(* IEC 61131-3 sources: st2cpp/tests/st_samples, 5 files *)

(* ---- test_array.st ---- *)
// ============================================================================
// ENUM Definitions
// ============================================================================

TYPE Color :
    (
    Red,
    Green := 5,
    Blue,
    Yellow := 10
    );
END_TYPE

TYPE Status :
    (
    Idle := 0,
    Running := 1,
    Stopped := 2,
    Error := 3
    );
END_TYPE

// ============================================================================
// STRUCT Definitions
// ============================================================================

TYPE Point3D :
    STRUCT
        x : INT;
        y : INT;
        z : INT;
    END_STRUCT
END_TYPE

TYPE MathEmbedded :
    STRUCT
        MathProcessor_ : MathProcessor;
        Point3D_ : Point3D;
    END_STRUCT
END_TYPE

TYPE struWithFB :
    STRUCT
        tryStruct : MathEmbedded;
    END_STRUCT
END_TYPE

TYPE Matrix3x3 :
    STRUCT
        data : ARRAY[1..3, 1..3] OF INT;  // 2D array inside struct
    END_STRUCT
END_TYPE

TYPE MultiArrayStruct :
    STRUCT
        arr1d : ARRAY[0..4] OF INT;
        arr2d : ARRAY[1..3, 0..2] OF INT;  // 3x3 matrix
        arr3d : ARRAY[0..1, 2..3, 0..2] OF REAL;  // 2x2x3 cube
    END_STRUCT
END_TYPE

// ============================================================================
// Function Block Definitions
// ============================================================================

FUNCTION_BLOCK MathProcessor
    VAR_INPUT
        a : INT;
        b : INT;
    END_VAR

    VAR_OUTPUT
        sum : INT;
        product : INT;
    END_VAR

    VAR
        temp : INT;
    END_VAR

    VAR_TEMP
        local_calc : INT;
    END_VAR

    METHOD Add : INT
        VAR_INPUT
            x : INT;
            y : INT;
        END_VAR
        Add := x + y;
    END_METHOD

    METHOD Multiply : INT
        VAR_INPUT
            x : INT;
            y : INT;
        END_VAR
        Multiply := x * y;
    END_METHOD
END_FUNCTION_BLOCK

// ============================================================================
// Global Variables with Arrays
// ============================================================================

VAR_GLOBAL
    // 1D arrays
    simple_array : ARRAY[0..5] OF INT := [10, 20, 30, 40, 50, 60];
    color_array : ARRAY[1..3] OF Color := [Color.Red, Color.Green, Color.Blue];
    empty_array : ARRAY[-2..2] OF REAL;

    // 2D arrays
    matrix_2x3 : ARRAY[0..1, 0..2] OF INT := [[1, 2, 3], [4, 5, 6]];
    identity_3x3 : ARRAY[1..3, 1..3] OF INT := [[1, 0, 0], [0, 1, 0], [0, 0, 1]];

    // 3D arrays
    cube_2x2x2 : ARRAY[0..1, 0..1, 0..1] OF INT;
    tensor : ARRAY[1..2, 2..3, 0..1] OF REAL := [[[1.1, 2.2], [3.3, 4.4]], [[5.5, 6.6], [7.7, 8.8]]];

    // Arrays of structs
    points : ARRAY[0..2] OF Point3D;

    // Arrays of function blocks
    processors : ARRAY[1..2] OF MathProcessor;

    // Complex nested arrays
    nested_array : ARRAY[0..1, 0..2] OF ARRAY[0..1] OF INT;  // Array of arrays
END_VAR

// ============================================================================
// Functions with Array Parameters
// ============================================================================

FUNCTION SumArray : INT
    VAR_INPUT
        arr : ARRAY[0..4] OF INT;
    END_VAR
    VAR
        i : INT;
        result : INT;
    END_VAR

    result := 0;
    FOR i := 0 TO 4 DO
        result := result + arr[i];
    END_FOR
    SumArray := result;
END_FUNCTION

FUNCTION MatrixMultiply : INT
    VAR_INPUT
        A : ARRAY[1..2, 1..2] OF INT;
        B : ARRAY[1..2, 1..2] OF INT;
        row : INT;
        col : INT;
    END_VAR
    VAR
        k : INT;
        result : INT;
    END_VAR

    result := 0;
    FOR k := 1 TO 2 DO
        result := result + A[row][k] * B[k][col];
    END_FOR
    MatrixMultiply := result;
END_FUNCTION

// ============================================================================
// Main Program
// ============================================================================

PROGRAM Main
    VAR
        counter : INT;
        statusVar : Status;
        colorVar : Color;
        point : Point3D;
        result : INT;
        i, j, k : INT;
        mat : ARRAY[1..3, 1..3] OF INT;
        cube : ARRAY[0..1, 0..1, 0..1] OF INT;
        proc : MathProcessor;
        mstruct : MultiArrayStruct;
    END_VAR

    // Test 1D arrays
    counter := simple_array[0] + simple_array[5];
    simple_array[2] := 100;
    empty_array[0] := 3.14;

    // Test enum arrays
    colorVar := color_array[2];
    IF colorVar = Color.Green THEN
        statusVar := Status.Running;
    END_IF

    // Test 2D arrays
    matrix_2x3[0][1] := 99;
    result := matrix_2x3[1][2];

    mat[1][1] := 10;
    mat[2][2] := 20;
    mat[3][3] := 30;

    // Test 3D arrays
    cube[0][0][0] := 1;
    cube[0][0][1] := 2;
    cube[1][1][1] := 8;

    // Nested loops for 3D array initialization
    FOR i := 0 TO 1 DO
        FOR j := 0 TO 1 DO
            FOR k := 0 TO 1 DO
                cube[i][j][k] := i * 100 + j * 10 + k;
            END_FOR
        END_FOR
    END_FOR

    // Test array initialization inside struct
    mstruct.arr1d[0] := 100;
    mstruct.arr2d[2][1] := 42;
    mstruct.arr3d[0][2][1] := 3.14159;

    // Test arrays of structs
    points[0].x := 10;
    points[1].y := 20;
    points[2].z := 30;

    // Test arrays of function blocks
    processors[1](a := 7, b := 4, sum => result);

    processors[2](a := 7, b := 4, product => result);

    // Test nested array access
    nested_array[0][1] := 42;

    // Complex array expressions
    simple_array[simple_array[0]] := 999;
    mat[counter][2] := simple_array[3];

    // Test multidimensional array in expression
    IF matrix_2x3[1][1] > 50 THEN
        statusVar := Status.Error;
    ELSE
        statusVar := Status.Stopped;
    END_IF

    // Test using MathProcessor methods
    proc( a := mat[1][1], b := mat[2][2], sum => result);

    // Test array bounds (will be checked in debug mode)
    // This would cause error in debug: simple_array[10] := 999;
END_PROGRAM

(* ---- test_inheritance.st ---- *)
// ============================================================================
// INTERFACES
// ============================================================================

INTERFACE I_Device
    METHOD Init : BOOL
        VAR_INPUT
            name : STRING;
        END_VAR
    END_METHOD

    METHOD GetName : STRING
    END_METHOD

    METHOD Process : BOOL
    END_METHOD

    METHOD GetStatus : INT
    END_METHOD
END_INTERFACE

INTERFACE I_Communicate
    METHOD Send : BOOL
        VAR_INPUT
            data : ARRAY[0..127] OF BYTE;
            len : INT;
        END_VAR
    END_METHOD

    METHOD Receive : BOOL
        VAR_OUTPUT
            data : ARRAY[0..127] OF BYTE;
            len : INT;
        END_VAR
    END_METHOD
END_INTERFACE

// ============================================================================
// ABSTRACT BASE CLASS
// ============================================================================

FUNCTION_BLOCK ABSTRACT FB_Device IMPLEMENTS I_Device
    VAR
        m_name : STRING;
        m_status : INT;
        m_errorCount : INT;
    END_VAR

    // Implementation of I_Device interface
    METHOD Init : BOOL
        VAR_INPUT
            name : STRING;
        END_VAR
        m_name := name;
        m_status := 0;
        m_errorCount := 0;
        Init := TRUE;
    END_METHOD

    METHOD GetName : STRING
        GetName := m_name;
    END_METHOD

    METHOD GetStatus : INT
        GetStatus := m_status;
    END_METHOD

    METHOD ABSTRACT Process : BOOL
    END_METHOD

    METHOD LogError
        VAR_INPUT
            errorCode : INT;
        END_VAR
        m_errorCount := m_errorCount + 1;
        m_status := errorCode;
    END_METHOD

    METHOD GetErrorCount : INT
        GetErrorCount := m_errorCount;
    END_METHOD
END_FUNCTION_BLOCK

// ============================================================================
// DERIVED CLASS - SENSOR
// ============================================================================

FUNCTION_BLOCK FB_Sensor EXTENDS FB_Device
    VAR
        m_value : REAL;
        m_threshold : REAL;
        m_sampleCount : INT;
    END_VAR

    METHOD OVERRIDE Process : BOOL
        Process := TRUE;
    END_METHOD

    METHOD SetThreshold
        VAR_INPUT
            threshold : REAL;
        END_VAR
        m_threshold := threshold;
    END_METHOD

    METHOD ReadValue : REAL
        ReadValue := m_value;
    END_METHOD

    METHOD Sample : BOOL
        VAR_INPUT
            newValue : REAL;
        END_VAR
        m_sampleCount := m_sampleCount + 1;
        m_value := newValue;

        IF m_value > m_threshold AND m_threshold > 0 THEN
            SUPER^.LogError(100);
            Sample := FALSE;
        ELSE
            Sample := TRUE;
        END_IF
    END_METHOD

    METHOD GetSampleCount : INT
        GetSampleCount := m_sampleCount;
    END_METHOD
END_FUNCTION_BLOCK

// ============================================================================
// DERIVED CLASS - ACTUATOR (FINAL - cannot be further inherited)
// ============================================================================

FUNCTION_BLOCK FINAL FB_Actuator EXTENDS FB_Device IMPLEMENTS I_Communicate
    VAR
        m_isRunning : BOOL;
        m_power : REAL;
        m_commandQueue : ARRAY[0..9] OF INT;
        m_queueHead : INT;
        m_queueTail : INT;
    END_VAR

    METHOD OVERRIDE Process : BOOL
        VAR
            i : INT;
        END_VAR
        Process := TRUE;
    END_METHOD

    METHOD Start : BOOL
        m_isRunning := TRUE;
        Start := TRUE;
    END_METHOD

    METHOD Stop : BOOL
        m_isRunning := FALSE;
        Stop := TRUE;
    END_METHOD

    METHOD SetPower
        VAR_INPUT
            powerPercent : REAL;
        END_VAR
        m_power := powerPercent;
    END_METHOD

    METHOD OVERRIDE LogError
        VAR_INPUT
            errorCode : INT;
        END_VAR
        // Override of LogError method
        SUPER^.LogError(errorCode);
        m_isRunning := FALSE;
    END_METHOD

    // Implementation of I_Communicate
    METHOD Send : BOOL
        VAR_INPUT
            data : ARRAY[0..127] OF BYTE;
            len : INT;
        END_VAR
        // Simulated command send
        Send := TRUE;
    END_METHOD

    METHOD Receive : BOOL
        VAR_OUTPUT
            data : ARRAY[0..127] OF BYTE;
            len : INT;
        END_VAR
        Receive := TRUE;
    END_METHOD

    METHOD QueueCommand
        VAR_INPUT
            cmd : INT;
        END_VAR
        m_commandQueue[m_queueTail] := cmd;
        m_queueTail := (m_queueTail + 1) MOD 10;
    END_METHOD

    METHOD ProcessQueue : BOOL
        VAR
            cmd : INT;
        END_VAR
        IF m_queueHead <> m_queueTail THEN
            cmd := m_commandQueue[m_queueHead];
            m_queueHead := (m_queueHead + 1) MOD 10;
            ProcessQueue := TRUE;
        ELSE
            ProcessQueue := FALSE;
        END_IF
    END_METHOD
END_FUNCTION_BLOCK

// ============================================================================
// DERIVED CLASS - TEMPERATURE SENSOR (SPECIALIZATION)
// ============================================================================

FUNCTION_BLOCK FB_TempSensor EXTENDS FB_Sensor
    VAR
        m_tempCelsius : REAL;
        m_offset : REAL;
    END_VAR

    METHOD OVERRIDE Process : BOOL
        VAR
            converted : REAL;
        END_VAR

        // Call base class Process method
        SUPER^.Process();

        // Convert Celsius to normalized value
        converted := (m_tempCelsius + m_offset) / 100.0;

        // Call base class Sample method (FB_Sensor)
        SUPER^.Sample(converted);

        Process := TRUE;
    END_METHOD

    METHOD SetTemperature
        VAR_INPUT
            celsius : REAL;
        END_VAR
        m_tempCelsius := celsius;
        m_value := celsius;  // m_value is defined in FB_Sensor
    END_METHOD

    METHOD SetOffset
        VAR_INPUT
            offset : REAL;
        END_VAR
        m_offset := offset;
    END_METHOD

    METHOD GetCelsius : REAL
        GetCelsius := m_tempCelsius + m_offset;
    END_METHOD
END_FUNCTION_BLOCK

// ============================================================================
// MAIN PROGRAM FOR TESTING
// ============================================================================

PROGRAM Main
    VAR
        // Direct instantiation
        sensor : FB_Sensor;
        actuator : FB_Actuator;
        tempSensor : FB_TempSensor;

        // Polymorphic array
        i : INT;

        // Test variables
        result : BOOL;
        name : STRING;
        status : INT;
        value : REAL;
        data : ARRAY[0..127] OF BYTE;
    END_VAR

    // ========================================================================
    // SENSOR TEST
    // ========================================================================

    // Initialization
    sensor.Init("TemperatureSensor");
    sensor.SetThreshold(50.0);

    // Method usage
    FOR i := 0 TO 9 DO
        sensor.Sample(i * 10.0);  // 0, 10, 20, 30, 40, 50...
    END_FOR

    status := sensor.GetStatus();
    value := sensor.ReadValue();
    name := sensor.GetName();
    result := sensor.Process();

    // ========================================================================
    // ACTUATOR TEST
    // ========================================================================

    actuator.Init("MotorController");
    actuator.Start();
    actuator.SetPower(75.0);
    actuator.QueueCommand(100);
    actuator.QueueCommand(200);
    result := actuator.ProcessQueue();

    // ========================================================================
    // TEMP SENSOR TEST (inheritance chain: FB_TempSensor -> FB_Sensor -> FB_Device)
    // ========================================================================

    tempSensor.Init("OvenSensor");
    tempSensor.SetThreshold(80.0);
    tempSensor.SetOffset(2.5);
    tempSensor.SetTemperature(75.0);

    result := tempSensor.Process();
    value := tempSensor.ReadValue();
    value := tempSensor.GetCelsius();
    status := tempSensor.GetErrorCount();

    // ========================================================================
    // SUPER^ TEST
    // ========================================================================

    // In tempSensor, Process calls SUPER^.Process() and SUPER^.Sample()
    // This verifies base-class call chaining

    // ========================================================================
    // FINAL CLASS TEST (FB_Actuator cannot be inherited)
    // ========================================================================

    // The following would cause a compile error:
    // FUNCTION_BLOCK FB_MyActuator EXTENDS FB_Actuator
    // END_FUNCTION_BLOCK
END_PROGRAM

(* ---- test_process_image.st ---- *)
(*
* test_process_image.st
* Test file for Process Image functionality
* Tests: %I, %Q, %M addresses with different qualifiers and placeholders "*"
*)

TYPE TestEnum :
    (
    IDLE,
    RUNNING,
    STOPPED,
    ERROR
    );
END_TYPE

TYPE MotorStatus :
    STRUCT
        Running : BOOL;
        Speed : INT;
        Temp : REAL;
        Fault : BOOL;
    END_STRUCT;
END_TYPE

(* Global variables with AT addresses - fixed and placeholder *)
VAR_GLOBAL
    (* Fixed addresses - will be marked as occupied *)
    StartButton AT %IX0.0 : BOOL := FALSE;
    StopButton AT %IX0.1 : BOOL := FALSE;
    Emergency AT %IX0.2 : BOOL := FALSE;

    MotorOutput AT %QX0.0 : BOOL := FALSE;
    AlarmLight AT %QX0.1 : BOOL := FALSE;
    StatusWord AT %QW2 : WORD := 16#0000;

    Counter AT %MW10 : INT := 0;
    Temperature AT %MW12 : INT := 25;
    Flags AT %MB20 : BYTE := 0;
    Status AT %ML22 : DWORD := 0;

    (* ========== PLACEHOLDER ADDRESSES - auto-allocated ========== *)

    (* BIT placeholders - will be allocated after fixed bits *)
    SensorA AT %IX* : BOOL := FALSE;       (* Will be allocated automatically *)
    SensorB AT %IX* : BOOL := FALSE;       (* Will be allocated automatically *)
    ActuatorA AT %QX* : BOOL := FALSE;     (* Will be allocated automatically *)
    ActuatorB AT %QX* : BOOL := FALSE;     (* Will be allocated automatically *)
    FlagA AT %MX* : BOOL := FALSE;         (* Will be allocated automatically *)

    (* BYTE placeholders - aligned to byte boundaries *)
    AnalogInput AT %IB* : BYTE := 0;       (* Will be allocated to %IB1 (after fixed bits) *)
    AnalogOutput AT %QB* : BYTE := 0;      (* Will be allocated automatically *)
    StatusFlags AT %MB* : BYTE := 0;       (* Will be allocated automatically *)

    (* WORD placeholders - must be aligned to 2-byte boundary *)
    Setpoint AT %IW* : INT := 100;         (* Will be allocated automatically *)
    Feedback AT %IW* : INT := 0;           (* Will be allocated automatically *)
    Command AT %QW* : WORD := 16#0000;     (* Will be allocated automatically *)
    MarkerData AT %MW* : WORD := 0;        (* Will be allocated automatically *)

    (* DWORD placeholders - must be aligned to 4-byte boundary *)
    LargeCounter AT %MD* : DWORD := 0;     (* Will be allocated automatically *)
    Timestamp AT %MD* : DWORD := 0;        (* Will be allocated automatically *)

    (* Mixed placeholders in different areas *)
    Diagnostic AT %MD* : DWORD := 0;       (* Will be allocated automatically *)
    DebugFlag AT %MX* : BOOL := FALSE;     (* Will be allocated automatically *)
    DebugValue AT %MW* : INT := 0;         (* Will be allocated automatically *)
END_VAR

(* Function block with process image access and methods *)
FUNCTION_BLOCK MotorController
    VAR_INPUT
        Enable : BOOL;
        Speed : INT;
    END_VAR

    VAR_OUTPUT
        Running : BOOL;
        Fault : BOOL;
    END_VAR

    VAR
        Timer : INT := 0;
        (* Local AT placeholder inside FB *)
        InternalFlag AT %MX* : BOOL := FALSE;  (* Will be allocated automatically *)
        InternalData AT %MW* : INT := 0;       (* Will be allocated automatically *)
    END_VAR

    METHOD CheckOverheat : BOOL
        VAR_INPUT
            Temp : INT;
        END_VAR
        VAR_OUTPUT
            Overheat : BOOL;
        END_VAR
        Overheat := Temp > 80;
        CheckOverheat := Overheat;
    END_METHOD

    METHOD ReadInternalData : INT
        VAR_OUTPUT
            Value : INT;
        END_VAR
        Value := InternalData;
    END_METHOD
END_FUNCTION_BLOCK

(* Main program - NO methods allowed! *)
PROGRAM Main
    VAR
        Motor : MotorController;
        TempRead : INT;
        State : TestEnum := TestEnum.IDLE;
        Status : MotorStatus;
        CycleCounter : INT := 0;
        NewState : TestEnum := IDLE;
        Updated : BOOL := FALSE;
        Start : BOOL := FALSE;
        Stop : BOOL := FALSE;
        EStop : BOOL := FALSE;
        Increment : BOOL := FALSE;
        NewTemp : INT := 0;
        (* Local AT placeholders inside program *)
        LocalSensor AT %IX* : BOOL := FALSE;   (* Will be allocated automatically *)
        LocalOutput AT %QX* : BOOL := FALSE;   (* Will be allocated automatically *)
        LocalData AT %MW* : INT := 0;          (* Will be allocated automatically *)
    END_VAR

    (* Main program body *)
    (* Read inputs *)
    Start := StartButton;
    Stop := StopButton;
    EStop := Emergency;

    (* Check emergency *)
    IF Emergency THEN
        MotorOutput := FALSE;
        AlarmLight := TRUE;
        Flags := Flags OR 16#80;
    END_IF;

    (* Update outputs based on state *)
    IF NOT Emergency THEN
        IF State = TestEnum.RUNNING THEN
            MotorOutput := TRUE;
            AlarmLight := FALSE;
            StatusWord := 16#0001;
        ELSIF State = TestEnum.STOPPED THEN
            MotorOutput := FALSE;
            AlarmLight := TRUE;
            StatusWord := 16#0002;
        ELSE
            MotorOutput := FALSE;
            AlarmLight := FALSE;
            StatusWord := 16#0000;
        END_IF;
    END_IF;

    (* Process counter *)
    IF Increment THEN
        Counter := Counter + 1;
    END_IF;

    (* Update temperature *)
    Temperature := NewTemp;
    Status.Temp := INT_TO_REAL(NewTemp) / 10.0;

    (* Use the function block *)
    Motor(Enable := Start, Speed := 100);

    (* Update status *)
    Updated := TRUE;

    (* Use local AT variables *)
    LocalSensor := SensorA;
    LocalOutput := ActuatorA;
    LocalData := Setpoint;
END_PROGRAM

(* Another program with different AT address patterns - NO methods! *)
PROGRAM Diagnostic
    VAR
        ErrorCode AT %MW50 : INT := 0;
        ErrorTime AT %MD52 : DWORD := 0;
        ErrorFlag AT %MX54.0 : BOOL := FALSE;
        Status AT %MW60 : INT := 0;
        Code : INT := 0;
        (* Local AT placeholders inside Diagnostic program *)
        DiagData AT %MD* : DWORD := 0;         (* Will be allocated automatically *)
        DiagFlag AT %MX* : BOOL := FALSE;      (* Will be allocated automatically *)
        DiagWord AT %MW* : WORD := 0;          (* Will be allocated automatically *)
    END_VAR

    (* Set error *)
    ErrorCode := Code;
    ErrorTime := 0;
    ErrorFlag := TRUE;
    Status := 1;

    (* Clear error *)
    ErrorCode := 0;
    ErrorTime := 0;
    ErrorFlag := FALSE;
    Status := 0;

    (* Use placeholders *)
    DiagData := ErrorTime;
    DiagFlag := ErrorFlag;
    DiagWord := 16#FFFF;
END_PROGRAM

(* Function that uses process image addresses - fixed and placeholder *)
FUNCTION GetMotorSpeed : INT
    VAR_INPUT
        MotorID : INT;
    END_VAR
    VAR
        Speed AT %IW100 : INT := 0;
        Speed2 AT %IW102 : INT := 0;
        (* Local AT placeholders inside function *)
        TempSpeed AT %IW* : INT := 0;          (* Will be allocated automatically *)
        SensorValue AT %IW* : INT := 0;        (* Will be allocated automatically *)
    END_VAR
    (* Read speed from input addresses *)
    IF MotorID = 1 THEN
        GetMotorSpeed := Speed;
    ELSE
        GetMotorSpeed := Speed2;
    END_IF;
END_FUNCTION

(* ---- test_program.st ---- *)
(*
* test_program.st
* Comprehensive test program for st2cpp generator
* Tests: FUNCTION_BLOCK with methods, FUNCTION calls, GVLs, ENUMs, STRUCTs, ARRAYs
*)

(* ============================================================================
*  ENUM definitions
* ============================================================================
*)

TYPE TestState :
    (
    IDLE,
    RUNNING,
    COMPLETED := 10,
    ERROR := 99
    );
END_TYPE

TYPE OperationMode :
    (
    MODE_AUTO,
    MODE_MANUAL,
    MODE_MAINTENANCE
    );
END_TYPE

(* ============================================================================
*  STRUCT definitions (simple, without FB)
* ============================================================================
*)
TYPE Point3D :
    STRUCT
        XY : Point2D;
        Z : INT := 0;
    END_STRUCT;
END_TYPE

TYPE Point2D :
    STRUCT
        X : INT := 0;
        Y : INT := 0;
    END_STRUCT;
END_TYPE

TYPE MathEmbedded :
    STRUCT
        MathProcessor_ : MathProcessor;
        Point3D_ : Point3D;
    END_STRUCT;
END_TYPE

TYPE struWithFB :
    STRUCT
        tryStruct : MathEmbedded;
    END_STRUCT
END_TYPE

(* ============================================================================
*  GLOBAL VARIABLES
* -============================================================================
*)

VAR_GLOBAL
    GlobalCounter : INT := 0;
    GlobalFlag : BOOL := FALSE;
    GlobalPosition : Point2D;
    GlobalArray : ARRAY [0..4] OF INT := [10, 20, 30, 40, 50];
END_VAR

(* ============================================================================
*  FUNCTIONS
* -============================================================================
*)

FUNCTION Add : INT
    VAR_INPUT
        A : INT;
        B : INT;
    END_VAR
    Add := A + B;
END_FUNCTION

FUNCTION Multiply : INT
    VAR_INPUT
        A : INT := 2;
        B : INT := 3;
    END_VAR
    VAR_OUTPUT
        Result : INT;
    END_VAR
    Result := A * B;
    Multiply := Result;
END_FUNCTION

FUNCTION ComplexCalc : REAL
    VAR_INPUT
        Input : INT;
        Multiplier : INT := 5;
    END_VAR
    VAR_OUTPUT
        Output : REAL;
        Status : BOOL;
    END_VAR
    VAR
        Temp : REAL;
    END_VAR
    Temp := Input * Multiplier;
    Output := Temp + 100.5;
    Status := Temp > 100.0;
    ComplexCalc := Output;
END_FUNCTION

(* ============================================================================
*  FUNCTION BLOCK with multiple methods
* -============================================================================
*)

FUNCTION_BLOCK MathProcessor
    VAR_INPUT
        Enable : BOOL;
        Factor : INT := 10;
    END_VAR
    VAR_OUTPUT
        Result : INT;
        IsBusy : BOOL;
        LastError : INT;
    END_VAR
    VAR
        InternalValue : INT := 0;
        OperationCount : INT := 0;
        ArrayBuffer : ARRAY [0..5] OF INT := [0, 1, 2, 3, 4, 5];
    END_VAR

    METHOD Reset : INT
        VAR_OUTPUT
            PreviousValue : INT;
        END_VAR
        PreviousValue := InternalValue;
        InternalValue := 0;
        OperationCount := 0;
        LastError := 0;
        Reset := PreviousValue;
    END_METHOD

    METHOD Process : INT
        VAR_INPUT
            Value : INT;
            Mode : OperationMode := OperationMode.MODE_AUTO;
        END_VAR
        VAR_OUTPUT
            ProcessedValue : INT;
            IsValid : BOOL;
        END_VAR
        VAR
            Temp : INT;
            Resukt : INT;
        END_VAR

        IF NOT Enable THEN
            LastError := -1;
            ProcessedValue := InternalValue;
            IsValid := FALSE;
            Process := InternalValue;
            RETURN;
        END_IF;

        OperationCount := OperationCount + 1;

        CASE Mode OF
            OperationMode.MODE_AUTO :
            Temp := Value * Factor;
            OperationMode.MODE_MANUAL :
            Temp := Value + InternalValue;
            OperationMode.MODE_MAINTENANCE :
            Temp := Value - Factor;
        END_CASE;

        InternalValue := InternalValue + Temp;
        ProcessedValue := InternalValue;
        IsValid := TRUE;
        Process := InternalValue;

        CASE value OF
            1, 3, 5:
                result := 1;
            10..20:
                result := 2;
            30..40, 50:
                result := 3;
            ELSE
                result := 0;
        END_CASE

        CASE value OF
            1, 3, 5:
                result := 1;
            10:
                result := 2;
            30, 40, 50:
                result := 3;
            ELSE
                result := 0;
        END_CASE

    END_METHOD

    METHOD GetStatistics : INT
        VAR_OUTPUT
            Count : INT;
            CurrentValue : INT;
            ArraySum : INT;
        END_VAR
        VAR
            I : INT;
        END_VAR
        Count := OperationCount;
        CurrentValue := InternalValue;
        ArraySum := 0;
        FOR I := 0 TO 5 DO
            ArraySum := ArraySum + ArrayBuffer[I];
        END_FOR;
        GetStatistics := ArraySum;
    END_METHOD

    METHOD AddToBuffer : BOOL
        VAR_INPUT
            Index : INT;
            Value : INT;
        END_VAR
        IF Index >= 0 AND Index <= 5 THEN
            ArrayBuffer[Index] := Value;
            AddToBuffer := TRUE;
        ELSE
            AddToBuffer := FALSE;
        END_IF;
    END_METHOD
END_FUNCTION_BLOCK

(* ============================================================================
*  FUNCTION BLOCK that uses another FB
* -============================================================================
*)

FUNCTION_BLOCK CompositeProcessor
    VAR_INPUT
        Enable : BOOL;
        InputValue : INT;
    END_VAR
    VAR_OUTPUT
        OutputValue : INT;
        StatusMessage : STRING;
    END_VAR
    VAR
        Math1 : MathProcessor;
        Math2 : MathProcessor;
        InternalState : TestState;
        CurrentPos : Point2D;
    END_VAR

    METHOD ProcessAll : INT
        VAR_OUTPUT
            Total : INT;
            Result1 : INT;
            Result2 : INT;
        END_VAR
        VAR
            Temp1 : INT;
            Temp2 : INT;
        END_VAR

        Math1.Enable := Enable;
        Math2.Enable := Enable;
        Math1.Factor := InputValue;
        Math2.Factor := InputValue * 2;

        Math1.Process(Value := InputValue, ProcessedValue => Temp1);
        Math2.Process(Value := InputValue * 2, ProcessedValue => Temp2);

        Result1 := Temp1;
        Result2 := Temp2;
        Total := Result1 + Result2;
        ProcessAll := Total;
    END_METHOD

    METHOD ResetAll : VOID
        Math1.Reset();
        Math2.Reset();
        InternalState := TestState.IDLE;
        CurrentPos.X := 0;
        CurrentPos.Y := 0;
    END_METHOD
END_FUNCTION_BLOCK

(* ============================================================================
*  PROGRAM Main
* -============================================================================
*)

PROGRAM MainTest
    VAR
        Processor : MathProcessor;
        Composite : CompositeProcessor;
        ResultValue : INT;
        Status : BOOL;
        CalcOutput : REAL;           // Per ComplexCalc Output
        CurrentVal : INT;            // Per GetStatistics CurrentValue
        ArraySumVal : INT;           // Per GetStatistics ArraySum
        TestArray : ARRAY [0..3] OF Point2D;
        CurrentMode : OperationMode;
        StateVar : TestState;
        ProcResult : INT;
        I : INT;
    END_VAR

    // Initialize
    Processor.Enable := TRUE;
    Processor.Factor := 5;
    Composite.Enable := TRUE;
    Composite.InputValue := 10;

    // Test method calls with various parameter styles
    Processor.Process(Value := 10, Mode := OperationMode.MODE_AUTO);
    Processor.Process(Value := 20);  // uses default MODE_AUTO
    Processor.Process(15, OperationMode.MODE_MANUAL);

    // Test function calls
    ResultValue := Add(25, 30);
    Multiply(Result := ResultValue);  // output binding
    ComplexCalc(Input := 100, Output => CalcOutput);  // CORRETTO

    // Test GetStatistics method
    Processor.GetStatistics(Count => ResultValue, CurrentValue => CurrentVal, ArraySum => ArraySumVal);  // CORRETTO

    // Test Reset method
    Processor.Reset(PreviousValue => ResultValue);

    // Test CompositeProcessor
    Composite.ProcessAll(Total => ProcResult);

    // Test global variables
    GlobalCounter := GlobalCounter + 1;
    GlobalPosition.X := GlobalPosition.X + 10;
    GlobalArray[2] := GlobalArray[2] + 5;

    // Test enum assignments
    StateVar := TestState.COMPLETED;
    CurrentMode := OperationMode.MODE_MAINTENANCE;

    // Test array of structs
    TestArray[0].X := 100;
    TestArray[0].Y := 200;
    TestArray[1].X := 300;
    TestArray[1].Y := 400;

    // Test conditionals
    IF Processor.Result > 100 THEN
        Status := TRUE;
    ELSE
        Status := FALSE;
    END_IF;

    // Test loop
    FOR I := 1 TO 10 DO
        ResultValue := ResultValue + I;
    END_FOR;

    // While loop with method call inside
    WHILE ResultValue < 1000 DO
        Processor.Process(Value := ResultValue);
        ResultValue := ResultValue + Processor.Result;
    END_WHILE;

END_PROGRAM

(* ---- library_usage.st ---- *)
// ============================================================================
// Uso di simboli provenienti dalle librerie esterne (examplelib + corelib):
//   - struct Channel (esterna, member Value/Limits: Limits e' corelib.Range)
//   - enum State (esterna) con enumeratori qualificati / non qualificati
//   - function Clamp (esterna, 3 parametri IN, ultimi due con default)
//   - FB TON (esterno, IN/PT e uscite Q/ET)
//   - constant MAX_CHANNELS (esterna)
//   - global gSystemState (esterna)
// ============================================================================

PROGRAM Main
    VAR
        ch : Channel;
        st : State;
        ton : TON;
        x : REAL;
        n : INT;
        done : BOOL;
        elapsed : TIME;
    END_VAR

    ch.Value := 8.5;
    ch.Limits.Min := 0.0;
    ch.Limits.Max := 10.0;

    st := State.FAULT;
    IF st = State.RUNNING THEN
        st := IDLE;
    END_IF

    x := Clamp(1.5, 0.0, 10.0);

    ton(IN := TRUE, PT := T#1s, Q => done, ET => elapsed);

    n := MAX_CHANNELS;
    st := gSystemState;
END_PROGRAM
